TYPE Rec_Other :
	STRUCT
		Compress_Home_Offset		:LREAL;
		Pusher_Home_Offset			:LREAL;
		Shield_Home_Offset			:LREAL;
		Axis_Acceleration			:LREAL;
		Axis_Deceleration			:LREAL;
		Axis_Jerk					:LREAL;
	END_STRUCT
END_TYPE

(* stored: Version 1.1.0.1, ProductVersion 3.1.4020.12
   DUT Rec_Other: Id {a72682aa-5a6c-4443-9fb6-6ddc66b23290} *)
